Fanuc KAREL source: compact_preamble.KL

PROGRAM KB00163
%NOLOCKGROUP
VAR
P1 : FILE
P2:INTEGER
BEGIN
P2=1
SET_FILE_ATR(P1,P2,1)
END KB00163
